// TIA Portal V16 export
// export: Created 2023-08-28T09:37:55.7208199Z, ExportSetting WithDefaults, DisplayName Totally Integrated Automation Portal, DisplayVersion V16 Update 6, DisplayName TIA Portal Version Control Interface, DisplayVersion V16 Update 2, DisplayName TIA Portal Openness, DisplayVersion V16 Update 6, DisplayName STEP 7 Professional, DisplayVersion V16 Update 6, DisplayName STEP 7 Safety, DisplayVersion V16, DisplayName WinCC Advanced, DisplayVersion V16 Update 6
VAR_GLOBAL   // PLC tag table "Sterowanie"
   INPUTstopAccident_Pompy AT %M84.3 : Bool;
   inputpowerOK_RS AT %M84.0 : Bool;
   "inputRem_P1-P4" AT %M84.1 : Bool;   // flaga tryb pracy zdalna / Tryb pracy 1=Auto, 0= Remontowe
   CMD_start_stop_inverter AT %M84.5 : Bool;   //    {ExternalWritable false}
   memRis_Foult_WiCC_PLC AT %M16.1 : Bool;   // Pamięć zbocza alarmu komunikacji WinCC-PLC
   memRis_WatchDog_HMI_PLC AT %M16.0 : Bool;   // Pamieć zbocza alarmu komunikacji KMI - PLC
   IsRem AT %M10.3 : Bool;   // Potwierdzenie trybu pracpomp 1=Auto, 0=Remontowe
   IsReady_Inverter AT %M10.7 : Bool;   // Znacznik gotowości falownika
   Mem_setMotor2 AT %M217.3 : Bool;   // Bit pamięci ustawienia pierwszego kompresora dodatkowego
   Mem_setMotor3 AT %M217.4 : Bool;   // Bit pamięci ustawienia drugiego kompresora dodatkowego
   mem_is_K1 AT %M218.1 : Bool;   // pamięć załaczenie znacznika pierwszej dodatkowego kompresora
   mem_Is_K2 AT %M218.2 : Bool;   // pamięć załaczenie znacznika pierwszej dodatkowego kompresora
   mem_Is_K3 AT %M218.3 : Bool;   // pamięć załaczenie znacznika wiodącego kompresora
   Is_extras_K1 AT %M219.2 : Bool;   // Znacznik dodatkowa 1
   Is_extras_K2 AT %M219.3 : Bool;   // Znacznik dodatkowa 2
   Is_up_Hz AT %M219.4 : Bool;   // Hz na wyjściu większe od minimalnych
   Mem_Res_setCMD_M9 AT %M11.7 : Bool;   // Pamięć zbocza blokowania stycznika falownik
   step_Hz_manual AT %MW26 : Int;   // Zmienna kroku ładowania Hz w trybie manual
   BarPress_Max AT %M219.6 : Bool;
   Set_50Hz AT %M219.7 : Bool;   // Znacznik pomocniczy dla procedury miękiego przełączenia Hz na falowniku
   mem_Triger_PowerOK AT %M220.0 : Bool;   // pamięć zbocza powroru zasilania
   Reset_HWork_errer AT %M220.1 : Bool;   // Kasowanie błędu ustawiania znaczników pracy od czasu
   Tmp_Set_SV AT %M220.4 : Bool;   // Znacznik ustawiania tymczasowej wartości Hz
   Rst_Driver_Max_presure AT %M221.6 : Bool;   // Znacznika awaryjnego wyłączenia od max ciśnienia napędu pracującego w trybie awaryjnym
   Switch_set_OverCurrentInverer AT %M10.0 : Bool;   // Przełącznik wyboru źródła zadawania wartości granicznej dopuszczalnego prądy falownika
   memZboczeN_wylK1 AT %M1101.0 : Bool;   // pamięć zbocza opadającego wyłaczenie dodatkowego 1
   srt50Hz_inverter_Level1 AT %M206.6 : Bool;   // Ustawienie 50 Hz w czasie wyłączenia dodatkowej Poziom 1
   isSetXXHz AT %M1101.1 : Bool;   // bit zatrzasku pamieci zboczaNeylK1
   RS_Zbocze_bar AT %M13.4 : Bool;   // Znacznik przekazujący info czy zbocze ciśnienieanarasta czy opada
   "inputready_Inverter_P1-P4" AT %M84.4 : Bool;   // gotowość faloenika
   Is_loading_K3 AT %M218.0 : Bool;   // Znacznik pompy wiodącej
   setPID_Pompy AT %M300.2 : Bool;   // Znacznik załączenie, regulacji falownika
   setMotor3 AT %M300.1 : Bool;   // Znacznik ustwienie dodatkowej dmuchawy nr2
   FC2_Set_50Hz AT %M15.0 : Bool;   // Zancznik ustalenia 50Hz
   Reset_Motor4_AlarmPresure AT %M90.2 : Bool;   // Znacznik wyłaczenia awaryjnego dmuchawy dodatkowej (alarm od ciśnienia)
   Reset_Motor4_AlarmOver AT %M90.3 : Bool;   // Znacznik wyłaczenia awaryjnego dmuchawy dodatkowej (alarm od przeciązenia)
   CMD_faultInverter AT %M90.4 : Bool;   // Znacznik awaria falownika
   CMD_faultP1 AT %M90.5 : Bool;   // Znacznik sygnalizacja awarii
   CMD_faultP2 AT %M90.6 : Bool;   // Znacznik sygnalizacja awarii
   CMD_faultP3 AT %M90.7 : Bool;   // Znacznik sygnalizacja awarii
   CMD_faultP4 AT %M91.0 : Bool;   // Znacznik sygnalizacja awarii
   setMotor4 AT %M300.6 : Bool;   // Znacznik ustwienie dodatkowej dmuchawy nr3
   memEdge_IsAut_pump AT %M19.1 : Bool;   // bit pamieci zbocza dla sygnału automatyczna praca pomp
   Mem_setMotor4 AT %M217.5 : Bool;   // Bit pamięci ustawienia trzeciej dodatkowej
   Is_extras_K3 AT %M221.7 : Bool;   // Znacznik dodatkowa 3
   memTrigSetAutomat AT %M19.2 : Bool;   // pamięć zbocza załaczenia trybu automat porzez stacyjki pomp
   memTrigManualFB1 AT %M19.7 : Bool;   // pamięć zbocza kontroli przełączników na HMI
   statMiasto AT %M54.0 : Bool;   // flaga start przetłaczanie - miasto
   statMagistrala AT %M54.1 : Bool;   // flaga start dosilanie - magistrala
   memTrigerStopAwariaPomp AT %M208.4 : Bool;   // pamięć zbocza dla zaczenia sygnalizacji wciśnięcia grzybka
   Reset_Motor3Alarm AT %M221.2 : Bool;   // Znacznik wyłączenia awaryjnego pompydodatkowej
   QW64 AT %QW64 : Int;   // Wartość Hz przekazywana na wyjście falownika
   inputrunInverter_ AT %M84.2 : Bool;   // Potwierdzenie załączeniea falownika
   Reset_Motor3_AlarmOver AT %M221.0 : Bool;   // Znacznik wyłaczenia awaryjnego pompy dodatkowej (alarm od ciśnienia)
   Reset_Motor3_AlarmPresure AT %M220.6 : Bool;   // Znacznik wyłaczenia awaryjnego pompydodatkowej (alarm od ciśnienia)
   IW166 AT %IW166 : Word;   // feedback act Hz
   Static_1 AT %MD222 : Real;
   IsCurrentOverloadInverter AT %M11.4 : Bool;   // Znacznik przeciążenie falownika kompresorów
   Reset_Motor2_AlarmPresure AT %M220.5 : Bool;   // Znacznik wyłaczenia awaryjnego pompydodatkowej (alarm od ciśnienia)
   Reset_Motor2Alarm AT %M221.1 : Bool;   // Znacznik wyłączenia awaryjnego pompy dodatkowej
   IsRunInverter1 AT %M211.2 : Bool;   // Potwierdzenie pracy falownika kompresorów
   IsModeAut AT %M12.3 : Bool;   // Flaga rozpoczęcia procedury sterowania automatycznego pompowni
   IW164 AT %IW164 : Word;   // poziom zbiornik nr3   {ExternalWritable false}
   ActCurrent_Supply_Inverter AT %MD212 : DWord;   // Aktualny prąd obciążenia falownika
   Reset_Motor2_AlarmOver AT %M220.7 : Bool;   // Znacznik wyłaczenia awaryjnego pompydodatkowej (alarm od ciśnienia)
   setMotor2 AT %M300.0 : Bool;   // Znacznik ustwienie dodatkowej dmuchawy nr1 / Znacznik ustwienie dodatkowej pompy nr1
   zbocze_dod_zegar AT %M93.7 : Bool;
   Is_PowerRS5_OK AT %M11.3 : Bool;   // Zasilanie RS Zasuwy
   is_Aut_Z9 AT %M84.6 : Bool;   // bit stausu automat zasuwy Z9
   Reset_Motor4Alarm AT %M90.1 : Bool;   // Znacznik wyłączenie od alarmu dodatkowej 3   {ExternalVisible false}
   FB9_Set_Motor3 AT %M220.3 : Bool;   // Znacznik dodatkowej pompy dla funkcji FB8 I / Znacznik dodakowapompa 2 dla funkcji FB8 I
   FB9_Set_Motor2 AT %M220.2 : Bool;   // Znacznik dodatkowej pompy dla funkcji FB8 I / Znacznik dodakowapompa 1 dla funkcji FB8 I
   FB9_Set_Motor4 AT %M300.5 : Bool;   // Znacznik dodatkowej pompy dla funkcji FB8 I / Znacznik dodakowapompa 3 dla funkcji FB8 I
END_VAR
